PROGRAM main
VAR
	S1 AT %IX0.0 : bool;
	S2 AT %IX0.1 : bool;
	H1 AT %QX0.0 : bool;
END_VAR

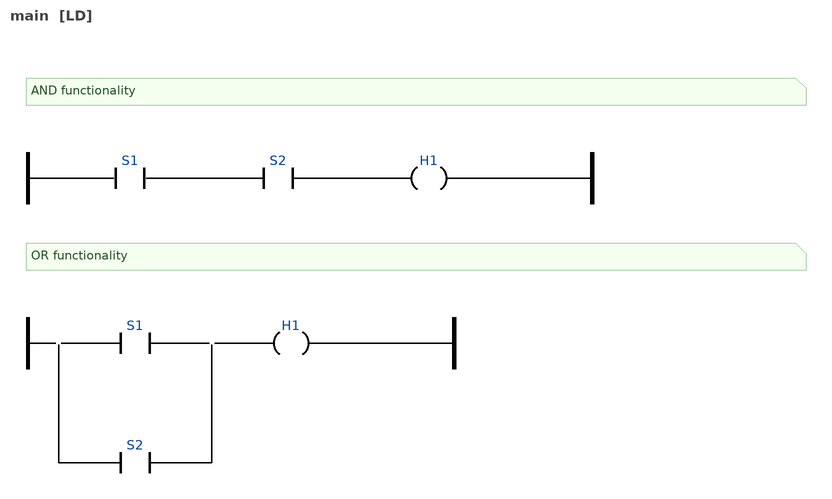
(* LD diagram, written out as Structured Text *)
(* AND functionality *)
H1 := S1 AND S2;
(* OR functionality *)
H1 := S1 OR S2;
END_PROGRAM
